# B&R Automation Studio project TD52 (part 19)

### mex.h
```c
/*
 * @(#)mex.h    generated by: makeheader 5.1.5  Tue May 24 21:10:37 2011
 *
 *		built from:	../../src/include/copyright.h
 *				../../src/include/pragma_interface.h
 *				mex_typedefs.h
 *				mexfunction.hpp
 *				fmexapi.cpp
 *				globals.cpp
 *				mexapi.cpp
 *				mexcbk.cpp
 *				mexdispatch.cpp
 *				mexintrf.cpp
 */

#if defined(_MSC_VER)
# pragma once
#endif
#if defined(__GNUC__) && (__GNUC__ > 3 || (__GNUC__ == 3 && __GNUC_MINOR__ > 3))
# pragma once
#endif

#ifndef mex_h
#define mex_h

/*
 * Copyright 1984-2003 The MathWorks, Inc.
 * All Rights Reserved.
 */

/* Copyright 2003-2006 The MathWorks, Inc. */

/* Only define EXTERN_C if it hasn't been defined already. This allows
 * individual modules to have more control over managing their exports.
 */
#ifndef EXTERN_C

#ifdef __cplusplus
  #define EXTERN_C extern "C"
#else
  #define EXTERN_C extern
#endif

#endif

/* Copyright 1999-2007 The MathWorks, Inc. */

/* $Revision: 1.7.4.4 $ */
#ifndef mex_typedefs_h
#define mex_typedefs_h

typedef struct impl_info_tag *MEX_impl_info;

#include "matrix.h"

#ifdef __cplusplus
extern "C"
{
#endif
typedef void (*mex_exit_fn)(void);
#ifdef __cplusplus
}
#endif

typedef struct mexGlobalTableEntry_Tag
{
    const char *name;             /* The name of the global */
    mxArray    **variable;        /* A pointer to the variable */
} mexGlobalTableEntry, *mexGlobalTable;

#ifdef _WIN32
#define cicompare(s1,s2) utStrcmpi((s1),(s2))
#else
#define cicompare(s1,s2) strcmp((s1),(s2))
#endif
#define cscompare(s1,s2) strcmp((s1),(s2))

typedef struct mexFunctionTableEntry_tag {
  const char *  name;
  mxFunctionPtr f;
  int           nargin;
  int           nargout;
  struct _mexLocalFunctionTable *local_function_table;
} mexFunctionTableEntry, *mexFunctionTable;

typedef struct _mexLocalFunctionTable {
  size_t           length;
  mexFunctionTable entries;
} _mexLocalFunctionTable, *mexLocalFunctionTable;

typedef struct {
  void (*initialize)(void);
  void (*terminate)(void);
} _mexInitTermTableEntry, *mexInitTermTableEntry;

#define MEX_INFORMATION_VERSION 1

typedef struct {
  int                   version;
  int                   file_function_table_length;
  mexFunctionTable      file_function_table;
  int                   global_variable_table_length;
  mexGlobalTable        global_variable_table;
  int                   npaths;
  const char **         paths;
  int                   init_term_table_length;
  mexInitTermTableEntry init_term_table;
} _mex_information, *mex_information;

typedef mex_information(*fn_mex_file)(void);

typedef void (*fn_clean_up_after_error)(void);
typedef const char *(*fn_simple_function_to_string)(mxFunctionPtr f);

typedef void (*fn_mex_enter_mex_library)(mex_information x);
typedef fn_mex_enter_mex_library fn_mex_exit_mex_library;

typedef mexLocalFunctionTable (*fn_mex_get_local_function_table)(void);
typedef mexLocalFunctionTable (*fn_mex_set_local_function_table)(mexLocalFunctionTable);

#endif

#ifdef DLL_EXPORT_SYM
# define MEXFUNCTION_LINKAGE EXTERN_C DLL_EXPORT_SYM
#else
# ifdef MW_NEEDS_VERSION_H
#  include "version.h"
#  define MEXFUNCTION_LINKAGE EXTERN_C DLL_EXPORT_SYM
# else
#  define MEXFUNCTION_LINKAGE EXTERN_C
# endif
#endif

MEXFUNCTION_LINKAGE
/*
 * mexFunction is the user-defined C routine that is called upon invocation
 * of a MEX-function.
 */
void mexFunction(
    int           nlhs,           /* number of expected outputs */
    mxArray       *plhs[],        /* array of pointers to output arguments */
    int           nrhs,           /* number of inputs */
    const mxArray *prhs[]         /* array of pointers to input arguments */
);

/*
 * This header file "mex.h" declares all the types, macros and
 * functions necessary to interface mex files with the current
 * version of MATLAB.  See the release notes for information on
 * supporting syntax from earlier versions.
 */
#include "matrix.h"

#include <stdio.h>

/*
 * Issue error message and return to MATLAB prompt
 */
EXTERN_C void mexErrMsgTxt(
    const char	*error_msg	/* string with error message */
    );

/*
 * Issue formatted error message with corresponding error identifier and return to MATLAB
 * prompt.
 */
EXTERN_C void mexErrMsgIdAndTxt(
    const char * identifier, /* string with error message identifier */
    const char * err_msg,    /* string with error message printf-style format */
    ...                      /* any additional arguments */
    );

/*
 * Invoke an unidentified warning. Such warnings can only be affected by the M-code
 * 'warning * all', since they have no specific identifier. See also mexWarnMsgIdAndTxt.
 */
EXTERN_C void mexWarnMsgTxt(
    const char	*warn_msg	/* string with warning message */
    );

/*
 * Invoke a warning with message identifier 'identifier' and message derived from 'fmt' and
 * subsequent arguments. The warning may either get printed as is (if it is set to 'on'), or
 * not actually get printed (if set to 'off'). See 'help warning' in MATLAB for more
 * details.
 */
EXTERN_C void mexWarnMsgIdAndTxt(
    const char * identifier,    /* string with warning message identifer */
    const char * warn_msg,	/* string with warning message printf-style format */
    ...                         /* any additional arguments */
    );

/*
 * mex equivalent to MATLAB's "disp" function
 */
EXTERN_C int mexPrintf(
    const char	*fmt,	/* printf style format */
    ...				/* any additional arguments */
    );

#define printf mexPrintf

/*
 * Remove all components of an array plus the array header itself
 * from MATLAB's memory allocation list.  The array will now
 * persist between calls to the mex function.  To destroy this
 * array, you will need to explicitly call mxDestroyArray().
 */
EXTERN_C void mexMakeArrayPersistent(
    mxArray *pa              /* pointer to array */
    );

/*
 * Remove memory previously allocated via mxCalloc from MATLAB's
 * memory allocation list.  To free this memory, you will need to
 * explicitly call mxFree().
 */
EXTERN_C void mexMakeMemoryPersistent(void *ptr);

/*
 * mex equivalent to MATLAB's "set" function
 */
EXTERN_C int mexSet(double handle, const char *property, mxArray *value);

/* API interface which mimics the "get" function */
EXTERN_C const mxArray *mexGet(double handle, const char *property);

/*
 * call MATLAB function
 */
EXTERN_C int mexCallMATLAB(
    int		nlhs,			/* number of expected outputs */
    mxArray	*plhs[],		/* pointer array to outputs */
    int		nrhs,			/* number of inputs */
    mxArray	*prhs[],		/* pointer array to inputs */
    const char	*fcn_name		/* name of function to execute */
    );

/*
 * call MATLAB function with Trap
 */
EXTERN_C mxArray	*mexCallMATLABWithTrap(
    int         nlhs,       /* number of expected outputs */
    mxArray     *plhs[],    /* pointer array to outputs */
    int         nrhs,       /* number of inputs */
    mxArray     *prhs[],    /* pointer array to inputs */
    const char  *fcn_name   /* name of function to execute */
    );

/*
 * set or clear mexCallMATLAB trap flag (if set then an error in
 * mexCallMATLAB is caught and mexCallMATLAB will return a status value,
 * if not set an error will cause control to revert to MATLAB)
 */
EXTERN_C void mexSetTrapFlag(int flag);

/*
 * Print an assertion-style error message and return control to the
 * MATLAB command line.
 */
EXTERN_C void mexPrintAssertion(
		const char *test,
		const char *fname,
		int linenum,
		const char *message);

/*
 * Tell whether or not a mxArray is in MATLAB's global workspace.
 */
EXTERN_C bool mexIsGlobal(const mxArray *pA);

/*
 * Place a copy of the array value into the specified workspace with the
 * specified name
 */
EXTERN_C int mexPutVariable(
    const char *workspace,
    const char *name,
    const mxArray *parray		/* matrix to copy */
    );

/*
 * return a pointer to the array value with the specified variable
 * name in the specified workspace
 */
EXTERN_C const mxArray *mexGetVariablePtr(
    const char *workspace,
    const char *name		/* name of symbol */
    );

/*
 * return a copy of the array value with the specified variable
 * name in the specified workspace
 */
EXTERN_C mxArray *mexGetVariable(
    const char	*workspace,
    const char  *name                /* name of variable in question */
    );

/*
 * Lock a MEX-function so that it cannot be cleared from memory.
 */
EXTERN_C void mexLock(void);

/*
 * Unlock a locked MEX-function so that it can be cleared from memory.
 */
EXTERN_C void mexUnlock(void);

/*
 * Return true if the MEX-function is currently locked, false otherwise.
 */
EXTERN_C bool mexIsLocked(void);

/*
 * Return the name of a the MEXfunction currently executing.
 */
EXTERN_C const char *mexFunctionName(void);

/*
 * Parse and execute MATLAB syntax in string.  Returns zero if successful,
 * and a non zero value if an error occurs.
 */
EXTERN_C int mexEvalString(
   const char *str	   /* matlab command string */
);

/*
 * Parse and execute MATLAB syntax in string.  Returns NULL if successful,
 * and an MException if an error occurs.
 */
EXTERN_C mxArray* mexEvalStringWithTrap(
   const char *str	   /* matlab command string */
);

/*
 * Register Mex-file's At-Exit function (accessed via MEX callback)
 */
EXTERN_C int mexAtExit(mex_exit_fn exit_fcn );

#endif /* mex_h */
```

### mwmathutil.h
```c
#if defined(_MSC_VER) || __GNUC__ > 3 || (__GNUC__ == 3 && __GNUC_MINOR__ > 3)
#pragma once
#endif

#ifndef mwmathutil_h
#define mwmathutil_h

/* Copyright 2003-2010 The MathWorks, Inc. */

/* Only define EXTERN_C if it hasn't been defined already. This allows
 * individual modules to have more control over managing their exports.
 */
#ifndef EXTERN_C

#ifdef __cplusplus
  #define EXTERN_C extern "C"
#else
  #define EXTERN_C extern
#endif

#endif

#include "tmwtypes.h"

/* abs(a) */
EXTERN_C double muDoubleScalarAbs(double a);

/* ceil(a) */
EXTERN_C double muDoubleScalarCeil(double a);

/* floor(a) */
EXTERN_C double muDoubleScalarFloor(double a);

/* round(a) */
EXTERN_C double muDoubleScalarRound(double a);

/* fix(a) */
EXTERN_C double muDoubleScalarFix(double xr);

/* acos(a) */
EXTERN_C double muDoubleScalarAcos(double a);

/* acosh(a) */
EXTERN_C double muDoubleScalarAcosh(double a);

/* asin(a) */
EXTERN_C double muDoubleScalarAsin(double a);

/* asinh(a) */
EXTERN_C double muDoubleScalarAsinh(double a);

/* atan(a) */
EXTERN_C double muDoubleScalarAtan(double a);

/* atanh(a) */
EXTERN_C double muDoubleScalarAtanh(double a);

/* cos(a) */
EXTERN_C double muDoubleScalarCos(double a);

/* cosh(a) */
EXTERN_C double muDoubleScalarCosh(double a);

/* exp(a) */
EXTERN_C double muDoubleScalarExp(double a);

/* log */
/*A warning 'Log of zero' should be issued by users for a = 0 */
EXTERN_C double muDoubleScalarLog(double a);

/* log10 */
/*A warning 'Log of zero' should be issued by users for a = 0 */
EXTERN_C double muDoubleScalarLog10(double a);

/* atan2(a,b) */
EXTERN_C double muDoubleScalarAtan2(double a, double b);

/* max(a,b) */
EXTERN_C double muDoubleScalarMax(double a, double b);

/* min(a,b) */
EXTERN_C double muDoubleScalarMin(double a, double b);

/* power(a,b) */
EXTERN_C double muDoubleScalarPower(double a, double b);

/* sin(a) */
EXTERN_C double muDoubleScalarSin(double a);

/* [s,c] = sincos(a) */
EXTERN_C void muDoubleScalarSinCos(double a, double* s, double* c);

/* sign(a) */
EXTERN_C double muDoubleScalarSign(double a);

/* sinh(a) */
EXTERN_C double muDoubleScalarSinh(double a);

/* sqrt(a) */
EXTERN_C double muDoubleScalarSqrt(double a);

/* tan(a) */
EXTERN_C double muDoubleScalarTan(double a);

/* tanh(a) */
EXTERN_C double muDoubleScalarTanh(double a);

/* mod(a,b) */
EXTERN_C double muDoubleScalarMod(double a, double b);

/* rem(a,b) */
EXTERN_C double muDoubleScalarRem(double a, double b);

/* hypot(a,b) */
EXTERN_C double muDoubleScalarHypot(double a,double b);

/* frexp(a,b) */
EXTERN_C double muDoubleScalarFrexp(double x, int *eptr);

/* abs(cmplx a) */
EXTERN_C double muDoubleComplexScalarAbs(double xr, double xi);

/* [br, bi] = exp(ar, ai) */
EXTERN_C void muDoubleComplexScalarExp(double *pyr, double *pyi, double xr, double xi);

/* hypot(ar, ai) */
EXTERN_C double muDoubleComplexScalarHypot(double ar, double ai, double br, double bi);

/* [br, bi] = log(ar, ai) */
EXTERN_C void muDoubleComplexScalarLog(double *pyr, double *pyi, double xr, double xi);

/* [cr, ci] = power(ar, ai, br, bi) */
EXTERN_C void muDoubleComplexScalarPower(double *cr, double *ci, double ar, double ai, double br, double bi);

/* [br, bi] = sqrt(ar, ai) */
EXTERN_C void muDoubleComplexScalarSqrt(double *br, double *bi, double ar, double ai);

/* [br, bi] = sign(ar, ai) */
EXTERN_C void muDoubleComplexScalarSign(double *br, double *bi, double ar, double ai);

/* [br, bi] = sin(ar, ai) */
EXTERN_C void muDoubleComplexScalarSin(double *br, double *bi, double ar, double ai);

/* [br, bi] = cos(ar, ai) */
EXTERN_C void muDoubleComplexScalarCos(double *br, double *bi, double ar, double ai);

/* [Sr, Si, Cr, Ci] = sincos(ar, ai) */
EXTERN_C void muDoubleComplexScalarSinCos(double *pySr, double *pySi, double *pyCr, double *pyCi,
                                          double xr, double xi);

/* [br, bi] = tan(ar, ai) */
EXTERN_C void muDoubleComplexScalarTan(double *br, double *bi, double ar, double ai);

/* [br, bi] = atan(ar, ai) */
EXTERN_C void muDoubleComplexScalarAtan(double *br, double *bi, double ar, double ai);

/* [br, bi] = asin(ar, ai) */
EXTERN_C void muDoubleComplexScalarAsin(double *br, double *bi, double ar, double ai);

/* [br, bi] = acos(ar, ai) */
EXTERN_C void muDoubleComplexScalarAcos(double *br, double *bi, double ar, double ai);

/* [br, bi] = sinh(ar, ai) */
EXTERN_C void muDoubleComplexScalarSinh(double *br, double *bi, double ar, double ai);

/* [br, bi] = cosh(ar, ai) */
EXTERN_C void muDoubleComplexScalarCosh(double *br, double *bi, double ar, double ai);

/* [br, bi] = tanh(ar, ai) */
EXTERN_C void muDoubleComplexScalarTanh(double *br, double *bi, double ar, double ai);

/* [br, bi] = asinh(ar, ai) */
EXTERN_C void muDoubleComplexScalarAsinh(double *br, double *bi, double ar, double ai);

/* [br, bi] = acosh(ar, ai) */
EXTERN_C void muDoubleComplexScalarAcosh(double *br, double *bi, double ar, double ai);

/* Single-precision functions */

/* abs(a) */
EXTERN_C float muSingleScalarAbs(float a);

/* ceil(a) */
EXTERN_C float muSingleScalarCeil(float a);

/* floor(a) */
EXTERN_C float muSingleScalarFloor(float a);

/* round(a) */
EXTERN_C float muSingleScalarRound(float a);

/* fix(a) */
EXTERN_C float muSingleScalarFix(float xr);

/* acos(a) */
EXTERN_C float muSingleScalarAcos(float a);

/* acosh(a) */
EXTERN_C float muSingleScalarAcosh(float a);

/* asin(a) */
EXTERN_C float muSingleScalarAsin(float a);

/* asinh(a) */
EXTERN_C float muSingleScalarAsinh(float a);

/* atan(a) */
EXTERN_C float muSingleScalarAtan(float a);

/* atanh(a) */
EXTERN_C float muSingleScalarAtanh(float a);

/* cos(a) */
EXTERN_C float muSingleScalarCos(float a);

/* cosh(a) */
EXTERN_C float muSingleScalarCosh(float a);

/* exp(a) */
EXTERN_C float muSingleScalarExp(float a);

/* log */
/*A warning 'Log of zero' should be issued by users for a = 0 */
EXTERN_C float muSingleScalarLog(float a);

/* log10 */
/*A warning 'Log of zero' should be issued by users for a = 0 */
EXTERN_C float muSingleScalarLog10(float a);

/* atan2(a,b) */
EXTERN_C float muSingleScalarAtan2(float a, float b);

/* max(a,b) */
EXTERN_C float muSingleScalarMax(float a, float b);

/* min(a,b) */
EXTERN_C float muSingleScalarMin(float a, float b);

/* power(a,b) */
EXTERN_C float muSingleScalarPower(float a, float b);

/* sin(a) */
EXTERN_C float muSingleScalarSin(float a);

/* [s,c] = sincos(a) */
EXTERN_C void muSingleScalarSinCos(float a, float* s, float* c);

/* sign(a) */
EXTERN_C float muSingleScalarSign(float a);

/* sinh(a) */
EXTERN_C float muSingleScalarSinh(float a);

/* sqrt(a) */
EXTERN_C float muSingleScalarSqrt(float a);

/* tan(a) */
EXTERN_C float muSingleScalarTan(float a);

/* tanh(a) */
EXTERN_C float muSingleScalarTanh(float a);

/* mod(a,b) */
EXTERN_C float muSingleScalarMod(float a, float b);

/* rem(a,b) */
EXTERN_C float muSingleScalarRem(float a, float b);

/* hypot(a,b) */
EXTERN_C float muSingleScalarHypot(float a,float b);

/* frexp(a,b) */
EXTERN_C float muSingleScalarFrexp(float x, int *eptr);

/* abs(cmplx a) */
EXTERN_C float muSingleComplexScalarAbs(float xr, float xi);

/* [br, bi] = exp(ar, ai) */
EXTERN_C void muSingleComplexScalarExp(float *pyr, float *pyi, float xr, float xi);

/* hypot(ar, ai) */
EXTERN_C float muSingleComplexScalarHypot(float ar, float ai, float br, float bi);

/* [br, bi] = log(ar, ai) */
EXTERN_C void muSingleComplexScalarLog(float *pyr, float *pyi, float xr, float xi);

/* [cr, ci] = power(ar, ai, br, bi) */
EXTERN_C void muSingleComplexScalarPower(float *cr, float *ci, float ar, float ai, float br, float bi);

/* [br, bi] = sqrt(ar, ai) */
EXTERN_C void muSingleComplexScalarSqrt(float *br, float *bi, float ar, float ai);

/* [br, bi] = sign(ar, ai) */
EXTERN_C void muSingleComplexScalarSign(float *br, float *bi, float ar, float ai);

/* [br, bi] = sin(ar, ai) */
EXTERN_C void muSingleComplexScalarSin(float *br, float *bi, float ar, float ai);

/* [br, bi] = cos(ar, ai) */
EXTERN_C void muSingleComplexScalarCos(float *br, float *bi, float ar, float ai);

/* [Sr, Si, Cr, Ci] = sincos(ar, ai) */
EXTERN_C void muSingleComplexScalarSinCos(float *pySr, float *pySi, float *pyCr, float *pyCi,
                                          float xr, float xi);

/* [br, bi] = tan(ar, ai) */
EXTERN_C void muSingleComplexScalarTan(float *br, float *bi, float ar, float ai);

/* [br, bi] = atan(ar, ai) */
EXTERN_C void muSingleComplexScalarAtan(float *br, float *bi, float ar, float ai);

/* [br, bi] = asin(ar, ai) */
EXTERN_C void muSingleComplexScalarAsin(float *br, float *bi, float ar, float ai);

/* [br, bi] = acos(ar, ai) */
EXTERN_C void muSingleComplexScalarAcos(float *br, float *bi, float ar, float ai);

/* [br, bi] = sinh(ar, ai) */
EXTERN_C void muSingleComplexScalarSinh(float *br, float *bi, float ar, float ai);

/* [br, bi] = cosh(ar, ai) */
EXTERN_C void muSingleComplexScalarCosh(float *br, float *bi, float ar, float ai);

/* [br, bi] = tanh(ar, ai) */
EXTERN_C void muSingleComplexScalarTanh(float *br, float *bi, float ar, float ai);

/* [br, bi] = asinh(ar, ai) */
EXTERN_C void muSingleComplexScalarAsinh(float *br, float *bi, float ar, float ai);

/* [br, bi] = acosh(ar, ai) */
EXTERN_C void muSingleComplexScalarAcosh(float *br, float *bi, float ar, float ai);

#ifdef __WATCOMC__
#pragma aux muDoubleScalarAbs value [8087];
#pragma aux muDoubleScalarCeil value [8087];
#pragma aux muDoubleScalarFloor value [8087];
#pragma aux muDoubleScalarRound value [8087];
#pragma aux muDoubleScalarAcos value [8087];
#pragma aux muDoubleScalarAcosh value [8087];
#pragma aux muDoubleScalarAsin value [8087];
#pragma aux muDoubleScalarAsinh value [8087];
#pragma aux muDoubleScalarAtan value [8087];
#pragma aux muDoubleScalarAtanh value [8087];
#pragma aux muDoubleScalarCos value [8087];
#pragma aux muDoubleScalarCosh value [8087];
#pragma aux muDoubleScalarExp value [8087];
#pragma aux muDoubleScalarLog value [8087];
#pragma aux muDoubleScalarLog10 value [8087];
#pragma aux muDoubleScalarAtan2 value [8087]
#pragma aux muDoubleScalarMax value [8087]
#pragma aux muDoubleScalarMin value [8087]
#pragma aux muDoubleScalarPower value [8087]
#pragma aux muDoubleScalarSin value [8087];
#pragma aux muDoubleScalarSinCos value [8087];
#pragma aux muDoubleScalarSign value [8087];
#pragma aux muDoubleScalarSinh value [8087];
#pragma aux muDoubleScalarSqrt value [8087];
#pragma aux muDoubleScalarTan value [8087];
#pragma aux muDoubleScalarTanh value [8087];
#pragma aux muDoubleScalarMod value [8087]
#pragma aux muDoubleScalarRem value [8087]
#pragma aux muDoubleScalarHypot value [8087];
#pragma aux muDoubleScalarFix value [8087];
#pragma aux muDoubleScalarFrexp value [8087];
#pragma aux muDoubleComplexScalarAbs value [8087];
#pragma aux muDoubleComplexScalarExp value [8087];
#pragma aux muDoubleComplexScalarHypot value [8087];
#pragma aux muDoubleComplexScalarLog value [8087];
#pragma aux muDoubleComplexScalarPower value [8087];
#pragma aux muDoubleComplexScalarSqrt value [8087];
#pragma aux muDoubleComplexScalarSign value [8087];
#pragma aux muDoubleComplexScalarSin value [8087];
#pragma aux muDoubleComplexScalarCos value [8087];
#pragma aux muDoubleComplexScalarSinCos value [8087];
#pragma aux muDoubleComplexScalarTan value [8087];
#pragma aux muDoubleComplexScalarAtan value [8087];
#pragma aux muDoubleComplexScalarAsin value [8087];
#pragma aux muDoubleComplexScalarAcos value [8087];
#pragma aux muDoubleComplexScalarSinh value [8087];
#pragma aux muDoubleComplexScalarCosh value [8087];
#pragma aux muDoubleComplexScalarTanh value [8087];
#pragma aux muDoubleComplexScalarAsinh value [8087];
#pragma aux muDoubleComplexScalarAcosh value [8087];
#pragma aux muSingleScalarAbs value [8087];
#pragma aux muSingleScalarCeil value [8087];
#pragma aux muSingleScalarFloor value [8087];
#pragma aux muSingleScalarRound value [8087];
#pragma aux muSingleScalarAcos value [8087];
#pragma aux muSingleScalarAcosh value [8087];
#pragma aux muSingleScalarAsin value [8087];
#pragma aux muSingleScalarAsinh value [8087];
#pragma aux muSingleScalarAtan value [8087];
#pragma aux muSingleScalarAtanh value [8087];
#pragma aux muSingleScalarCos value [8087];
#pragma aux muSingleScalarCosh value [8087];
#pragma aux muSingleScalarExp value [8087];
#pragma aux muSingleScalarLog value [8087];
#pragma aux muSingleScalarLog10 value [8087];
#pragma aux muSingleScalarAtan2 value [8087]
#pragma aux muSingleScalarMax value [8087]
#pragma aux muSingleScalarMin value [8087]
#pragma aux muSingleScalarPower value [8087]
#pragma aux muSingleScalarSin value [8087];
#pragma aux muSingleScalarSinCos value [8087];
#pragma aux muSingleScalarSign value [8087];
#pragma aux muSingleScalarSinh value [8087];
#pragma aux muSingleScalarSqrt value [8087];
#pragma aux muSingleScalarTan value [8087];
#pragma aux muSingleScalarTanh value [8087];
#pragma aux muSingleScalarMod value [8087]
#pragma aux muSingleScalarRem value [8087]
#pragma aux muSingleScalarHypot value [8087];
#pragma aux muSingleScalarFix value [8087];
#pragma aux muSingleScalarFrexp value [8087];
#pragma aux muSingleComplexScalarAbs value [8087];
#pragma aux muSingleComplexScalarExp value [8087];
#pragma aux muSingleComplexScalarHypot value [8087];
#pragma aux muSingleComplexScalarLog value [8087];
#pragma aux muSingleComplexScalarPower value [8087];
#pragma aux muSingleComplexScalarSqrt value [8087];
#pragma aux muSingleComplexScalarSign value [8087];
#pragma aux muSingleComplexScalarSin value [8087];
#pragma aux muSingleComplexScalarCos value [8087];
#pragma aux muSingleComplexScalarSinCos value [8087];
#pragma aux muSingleComplexScalarTan value [8087];
#pragma aux muSingleComplexScalarAtan value [8087];
#pragma aux muSingleComplexScalarAsin value [8087];
#pragma aux muSingleComplexScalarAcos value [8087];
#pragma aux muSingleComplexScalarSinh value [8087];
#pragma aux muSingleComplexScalarCosh value [8087];
#pragma aux muSingleComplexScalarTanh value [8087];
#pragma aux muSingleComplexScalarAsinh value [8087];
#pragma aux muSingleComplexScalarAcosh value [8087];
#endif

/* Integer Scalar functions. */
/* Integer Abs Family. */
EXTERN_C uint8_T muIntScalarAbs_uint8(uint8_T a);

EXTERN_C int8_T muIntScalarAbs_sint8(int8_T a);

EXTERN_C uint16_T muIntScalarAbs_uint16(uint16_T a);

EXTERN_C int16_T muIntScalarAbs_sint16(int16_T a);

EXTERN_C uint32_T muIntScalarAbs_uint32(uint32_T a);

EXTERN_C int32_T muIntScalarAbs_sint32(int32_T a);

/* Integer Max Family. */
EXTERN_C uint8_T muIntScalarMax_uint8(uint8_T a, uint8_T b);

EXTERN_C int8_T muIntScalarMax_sint8(int8_T a, int8_T b);

EXTERN_C uint16_T muIntScalarMax_uint16(uint16_T a, uint16_T b);

EXTERN_C int16_T muIntScalarMax_sint16(int16_T a, int16_T b);

EXTERN_C uint32_T muIntScalarMax_uint32(uint32_T a, uint32_T b);

EXTERN_C int32_T muIntScalarMax_sint32(int32_T a, int32_T b);

/* Integer Min Family. */
EXTERN_C uint8_T muIntScalarMin_uint8(uint8_T a, uint8_T b);

EXTERN_C int8_T muIntScalarMin_sint8(int8_T a, int8_T b);

EXTERN_C uint16_T muIntScalarMin_uint16(uint16_T a, uint16_T b);

EXTERN_C int16_T muIntScalarMin_sint16(int16_T a, int16_T b);

EXTERN_C uint32_T muIntScalarMin_uint32(uint32_T a, uint32_T b);

EXTERN_C int32_T muIntScalarMin_sint32(int32_T a, int32_T b);

/* Integer Mod Family. */
EXTERN_C uint8_T muIntScalarMod_uint8(uint8_T a, uint8_T b);

EXTERN_C int8_T muIntScalarMod_sint8(int8_T a, int8_T b);

EXTERN_C uint16_T muIntScalarMod_uint16(uint16_T a, uint16_T b);

EXTERN_C int16_T muIntScalarMod_sint16(int16_T a, int16_T b);

EXTERN_C uint32_T muIntScalarMod_uint32(uint32_T a, uint32_T b);

EXTERN_C int32_T muIntScalarMod_sint32(int32_T a, int32_T b);

/* Integer Rem Family. */
EXTERN_C uint8_T muIntScalarRem_uint8(uint8_T a, uint8_T b);

EXTERN_C int8_T muIntScalarRem_sint8(int8_T a, int8_T b);

EXTERN_C uint16_T muIntScalarRem_uint16(uint16_T a, uint16_T b);

EXTERN_C int16_T muIntScalarRem_sint16(int16_T a, int16_T b);

EXTERN_C uint32_T muIntScalarRem_uint32(uint32_T a, uint32_T b);

EXTERN_C int32_T muIntScalarRem_sint32(int32_T a, int32_T b);

/* Integer Sign Family. */
EXTERN_C uint8_T muIntScalarSign_uint8(uint8_T a);

EXTERN_C int8_T muIntScalarSign_sint8(int8_T a);

EXTERN_C uint16_T muIntScalarSign_uint16(uint16_T a);

EXTERN_C int16_T muIntScalarSign_sint16(int16_T a);

EXTERN_C uint32_T muIntScalarSign_uint32(uint32_T a);

EXTERN_C int32_T muIntScalarSign_sint32(int32_T a);

/* isFinite(a) */
EXTERN_C boolean_T muDoubleScalarIsFinite(double a);

/* isNaN(a) */
EXTERN_C boolean_T muDoubleScalarIsNaN(double a);

/* isInf(a) */
EXTERN_C boolean_T muDoubleScalarIsInf(double a);

/* isFinite(ar, ai) */
EXTERN_C boolean_T muDoubleComplexScalarIsFinite(double ar, double ai);

/* isNaN(a) */
EXTERN_C boolean_T muDoubleComplexScalarIsNaN(double ar, double ai);

/* isInf(ar, ai) */
EXTERN_C boolean_T muDoubleComplexScalarIsInf(double ar, double ai);

/* Single-precision functions */

/* isFinite(a) */
EXTERN_C boolean_T muSingleScalarIsFinite(float a);

/* isNaN(a) */
EXTERN_C boolean_T muSingleScalarIsNaN(float a);

/* isInf(a) */
EXTERN_C boolean_T muSingleScalarIsInf(float a);

/* isFinite(ar, ai) */
EXTERN_C boolean_T muSingleComplexScalarIsFinite(float ar, float ai);

/* isNaN(a) */
EXTERN_C boolean_T muSingleComplexScalarIsNaN(float ar, float ai);

/* isInf(ar, ai) */
EXTERN_C boolean_T muSingleComplexScalarIsInf(float ar, float ai);

#endif /* mwmathutil_h */
```

### mwutil.h
```c
/*
 * @(#)mwutil.h    generated by: makeheader 5.1.5  Tue May 24 21:07:18 2011
 *
 *		built from:	../../src/include/copyright.h
 *				../../src/include/pragma_interface.h
 *				cputime.cpp
 *				cycles.cpp
 *				dconvert.cpp
 *				demangle.cpp
 *				dynload.cpp
 *				emptystr.cpp
 *				enum_str.cpp
 *				expmatch.cpp
 *				f2cstr.cpp
 *				fgets.cpp
 *				filelink.cpp
 *				format.cpp
 *				fp_conv.cpp
 *				fpu.cpp
 *				getcwd.cpp
 *				hash.cpp
 *				incrfcn.cpp
 *				int_conv.cpp
 *				logfile.cpp
 *				lower.cpp
 *				multibyte.cpp
 *				mwclasses.cpp
 *				perfcount.cpp
 *				printf.cpp
 *				purifytools.cpp
 *				set.cpp
 *				special_nans.cpp
 *				stacktrc.cpp
 *				strcat.cpp
 *				strcmp.cpp
 *				strcmpi.cpp
 *				strcpy.cpp
 *				strdup.cpp
 *				strlen.cpp
 *				strrep.cpp
 *				strrstr.cpp
 *				strtok.cpp
 *				sysinfo.cpp
 *				timeinfo.cpp
 *				tmpnam.cpp
 *				tolower.cpp
 *				upper.cpp
 *				utStreamUtilities.cpp
 *				ut_alloca.cpp
 *				utassert.cpp
 *				utcrc.cpp
 *				utsignal.cpp
 *				wallclok.cpp
 *				array/array.cpp
 *				basic/basic_contexts.cpp
 *				checksum/md5checksum.cpp
 *				coll/functional.cpp
 *				coll/hash_map.cpp
 *				coll/hashrank.cpp
 *				cpputils/attacher.cpp
 *				cpputils/chunkedptr.cpp
 *				cpputils/countlist.cpp
 *				cpputils/safepointer.cpp
 *				cpputils/stat_ref_ok.cpp
 *				cpputils/stl_allocator.cpp
 *				dsbuffer/dsbuffer.cpp
 *				dtoa/dtoa.cpp
 *				dtoa/fpc.cpp
 *				dtoa/g_fmt.cpp
 *				err/error_context.cpp
 *				except/cmnHooks.cpp
 *				except/cmnSystemCalls.cpp
 *				except/errInternalException.cpp
 *				except/errSystemError.cpp
 *				except/errThrowable.cpp
 *				except/errUserException.cpp
 *				except/exceptCleanup.cpp
 *				except/exceptTypedefs.cpp
 *				except/instCpuCounter.cpp
 *				except/instInstrument.cpp
 *				except/instStopwatch.cpp
 *				except/logBasicSystemHandler.cpp
 *				except/logDataOutput.cpp
 *				except/logDebugOutputHandler.cpp
 *				except/logExternalizable.cpp
 *				except/logFilter.cpp
 *				except/logFormattable.cpp
 *				except/logFormatter.cpp
 *				except/logHandler.cpp
 *				except/logLevel.cpp
 *				except/logLogger.cpp
 *				except/logObjectOutput.cpp
 *				except/logObjectOutputStream.cpp
 *				except/logOutputStreamHandler.cpp
 *				except/logStreamHandler.cpp
 *				except/logTerminalHandler.cpp
 *				except/logXmlFormatter.cpp
 *				except/msgMsgCodeException.cpp
 *				except/msgMsgFormat.cpp
 *				except/usrReport.cpp
 *				except/usrRunning.cpp
 *				except/usrStartup.cpp
 *				except/usrStrategy.cpp
 *				ghash/ghash.cpp
 *				gtable/gtable.cpp
 *				hashtool/hashtool.cpp
 *				icuext/uchar.cpp
 *				icuext/uconv.cpp
 *				icuext/uctype.cpp
 *				icuext/uerror.cpp
 *				icuext/uhash.cpp
 *				icuext/umisc.cpp
 *				icuext/urecognize.cpp
 *				icuext/uspecial.cpp
 *				icuext/ustdio.cpp
 *				icuext/ustring.cpp
 *				icuext/utf.cpp
 *				icuext/utf8str.cpp
 *				ihash/ihash.cpp
 *				interval/fsi.cpp
 *				lcctype/utctype.cpp
 *				linebuf/linebuf.cpp
 *				mem/memory_context.cpp
 *				memmgr/memalloc.cpp
 *				msg/message_context.cpp
 *				nh/namehash.cpp
 *				nh/symtab.cpp
 *				profile/profile.cpp
 *				regexp/re_api.cpp
 *				regexp/re_builder.cpp
 *				regexp/re_collection.cpp
 *				regexp/re_context.cpp
 *				regexp/re_evaluator.cpp
 *				regexp/re_flags.cpp
 *				regexp/re_memory.cpp
 *				regexp/re_node_factory.cpp
 *				regexp/re_parser.cpp
 *				regexp/re_parser_context.cpp
 *				regexp/re_private_nodes.cpp
 *				regexp/re_protected_nodes.cpp
 *				regexp/re_replace.cpp
 *				regexp/re_replace_nodes.cpp
 *				regexp/re_replace_parser.cpp
 *				regexp/re_replaceable.cpp
 *				regexp/re_results.cpp
 *				regexp/re_search_info.cpp
 *				regexp/re_token_info.cpp
 *				regexp/re_translate.cpp
 *				regexp/re_tree.cpp
 *				regexp/re_tree_parser.cpp
 *				regexp/re_util.cpp
 *				sort/qsort.cpp
 *				strbuf/string_buffer.cpp
 *				threads/atomic.cpp
 *				threads/mwatomic.cpp
 *				threads/mwbarrier.cpp
 *				threads/mwconcurrent.cpp
 *				threads/mwcondition.cpp
 *				threads/mwcountedbody.cpp
 *				threads/mwcountedpointer.cpp
 *				threads/mwevent.cpp
 *				threads/mwmonitor.cpp
 *				threads/mwmutex_lwm.cpp
 *				threads/mwmutexlock.cpp
 *				threads/mwobjmgr.cpp
 *				threads/mwpointer.cpp
 *				threads/mwrcrsvmtx.cpp
 *				threads/mwsemaphore.cpp
 *				threads/mwsingleton.cpp
 *				threads/mwthdspc.cpp
 *				threads/mwthread.cpp
 *				threads/mwthreadid.cpp
 *				threads/mwtimeunit.cpp
 *				threads/ut_thread.cpp
 *				tse/tse.cpp
 *				warn/warning_context.cpp
 *				warn/warnmgr.cpp
 */

#if defined(_MSC_VER)
# pragma once
#endif
#if defined(__GNUC__) && (__GNUC__ > 3 || (__GNUC__ == 3 && __GNUC_MINOR__ > 3))
# pragma once
#endif

#ifndef mwutil_h
#define mwutil_h

/*
 * Copyright 1984-2003 The MathWorks, Inc.
 * All Rights Reserved.
 */

/* Copyright 2003-2006 The MathWorks, Inc. */

/* Only define EXTERN_C if it hasn't been defined already. This allows
 * individual modules to have more control over managing their exports.
 */
#ifndef EXTERN_C

#ifdef __cplusplus
  #define EXTERN_C extern "C"
#else
  #define EXTERN_C extern
#endif

#endif

/*
 * load library into memory
 */
EXTERN_C void *utLoadLibrary(
    const char	*fullname,	/* _full_ library path name */
    int		*errorStatus	/* return variable for error code */
    );

/*
 * Check whether shared library is loaded without loading it
 * Takes basename. Returns true if the library is loaded
 */
EXTERN_C bool utIsLibraryLoaded(const char *name);

/*
 * Return handle for already loaded library
 */
EXTERN_C void *utLoadModule(const char *basename);

/*
 * lookup symbol in a loaded library
 */
EXTERN_C void *utFindSymbolInLibrary(
    void        *handle,	/* handle returned by utLoadLibrary */
    const char  *symbol         /* symbol name to look up */
    );

/*
 * unload a previously loaded library
 */
EXTERN_C int utUnloadLibrary(
    void        *handle		/* handle returned by utLoadLibrary */
    );

/*
 * Retrieve last error in dynamic loader utility routines
 */
EXTERN_C const char *utLastLibraryError(void);

/*
 * Predicate to determine whether a double is an int.
 * -0 is not considered an int, because converting it back
 * does not yield the same double.
 */
EXTERN_C bool utDblIsInt(double x);

/*
 * Use unique NaNs as flags for special values
 * These values should never be generated by Matlab as valid NaNs.
 *
 * The low-order word is all zeros.
 */

#define UT_SPECIAL_NAN 0x7ff5c5c0

#define UT_NAN_NEVER_TOUCHED (UT_SPECIAL_NAN + 0x1)
#define UT_NAN_FORLOOP_EMPTY (UT_SPECIAL_NAN + 0x2)

#define UT_SET_NAN_VALUE(lval, jqnan) ut_SET_BOTH(lval, jqnan, 0)

/*
 * since the x86 fpu can change the leading mastissa bit on QNaNs, we check for
 * equality with and without the bit set.
 */
#define UT_QNAN_BITMASK 0x00080000
#define UT_IS_NAN_VALUE(val, jqnan)                                                                     \
    (*(((int*)&(val))+(CPU_NUM_FORMAT==FIEEE_BE)) == 0x0 &&                                             \
     (*(((int*)&(val))+(CPU_NUM_FORMAT==FIEEE_LE))|UT_QNAN_BITMASK) == ((jqnan)|UT_QNAN_BITMASK))

# define utAssert(test)             ((void)0)
# define utAssertStr(test, message) ((void)0)
# define utAssertAlways(message)    ((void)0)

#endif /* mwutil_h */
```

### odesup.h
```c
/*
 * Copyright 1994-2008 The MathWorks, Inc.
 *
 * File: odesup.h     $Revision: 1.3.4.3 $
 *
 * Abstract:
 *
 */

#ifndef __ODE_SUP__
#define __ODE_SUP__

#include <math.h>
#include <stddef.h> /* needed for NULL */

#include "tmwtypes.h"

#ifdef RT_MALLOC
# include <stdlib.h>
#endif

#ifdef USE_RTMODEL
# include "simstruc_types.h"
#else
# include "simstruc.h"
#endif

#ifndef RT_MALLOC
# ifndef NCSTATES
#  error "must define NCSTATES"
# endif
#endif

extern const char *RT_MEMORY_ALLOCATION_ERROR;

#ifdef RT_MALLOC
# define DERIVATIVES(si) rtmiDerivatives(*rtsiGetModelMethodsPtr(si))
# define PROJECTION(si)  rtmiProjection(*rtsiGetModelMethodsPtr(si))
# define OUTPUTS(si,tid) rtmiOutputs(*rtsiGetModelMethodsPtr(si),tid)
#else
# define DERIVATIVES(si) MdlDerivatives()
# define OUTPUTS(si,tid) MdlOutputs(tid)
# define PROJECTION(si)  MdlProjection()
  extern void MdlDerivatives(void);
  extern void MdlOutputs(int_T tid);
  extern void MdlProjection(void);
#endif

#ifndef USE_RTMODEL

void rt_ODECreateIntegrationData(RTWSolverInfo *si);
void rt_ODEDestroyIntegrationData(RTWSolverInfo *si);
void rt_ODEUpdateContinuousStates(RTWSolverInfo *si);

void rt_ODECacheDataIntoSolverInfo(SimStruct *S)
{
    RTWSolverInfo *si = ssGetRTWSolverInfo(S);

    if (si != NULL) {
        rtsiSetSolverStopTime(si, ssGetSolverStopTime(S));
        rtsiSetSolverName(si, ssGetSolverName(S));
        rtsiSetSolverData(si, ssGetSolverData(S));
    }
}

void rt_ODERetrieveDataFromSolverInfo(SimStruct *S)
{
    RTWSolverInfo *si = ssGetRTWSolverInfo(S);

    if (si != NULL) {
        ssSetSolverStopTime(S, rtsiGetSolverStopTime(si));
        ssSetSolverData(S, rtsiGetSolverData(si));
        ssSetSolverName(S, rtsiGetSolverName(si));
    }
}

const char_T *rt_ODECreateSolverInfo(SimStruct *S)
{
    const char_T          *errStatus = NULL;
    RTWSolverInfo         *si        = NULL;
    RTWRTModelMethodsInfo *mmi       = NULL;

#ifndef RT_MALLOC
    static RTWSolverInfo _si;
    static RTWRTModelMethodsInfo _mdlMths;

    si  = &_si;
    mmi = &_mdlMths;
#else
    si = (RTWSolverInfo *)malloc(sizeof(RTWSolverInfo));
    if (si == NULL) {
        errStatus = RT_MEMORY_ALLOCATION_ERROR;
        ssSetErrorStatus(S, RT_MEMORY_ALLOCATION_ERROR);
        goto EXIT_POINT;
    }

    mmi = (RTWRTModelMethodsInfo *)malloc(sizeof(RTWRTModelMethodsInfo));
    if (mmi == NULL) {
        errStatus = RT_MEMORY_ALLOCATION_ERROR;
        ssSetErrorStatus(S, RT_MEMORY_ALLOCATION_ERROR);
        goto EXIT_POINT;
    }
#endif

    rtsiSetModelMethodsPtr(si, mmi);
    rtsiSetRTModelPtr(si, (void *)S);
    rtmiSetRTModelPtr(*mmi, (void *)S);

    ssSetRTWSolverInfo(S, si);

    /*
     * The fields below need to be copied over at setup
     * and copied back into the SimStruct at the end
     */
    rt_ODECacheDataIntoSolverInfo(S);

    /*
     * The fields below only need to be setup. They are
     * pointer fields and updating them will automatically
     * update the owner SimStruct
     */

    /* Copy over a pointer to StepSize */
    rtsiSetStepSizePtr(si, &ssGetStepSize(S));

    /* Copy over a pointer to SimTimeStep */
    rtsiSetSimTimeStepPtr(si, &ssGetSimTimeStep(S));

    /* Copy over a pointer to the time pointer */
    rtsiSetTPtr(si, &ssGetTPtr(S));

    /* Copy over a pointer to the location of the derivs */
    rtsiSetdXPtr(si, &ssGetdX(S));

    /* Copy over a pointer to the location of the cont states */
    rtsiSetContStatesPtr(si, &ssGetContStates(S));

    /* Copy over a pointer to the location of the number of cont states */
    rtsiSetNumContStatesPtr(si, &ssGetNumContStates(S));

    /* Copy over a pointer to the location of the error status */
    rtsiSetErrorStatusPtr(si, &ssGetErrorStatus(S));

    /* Copy over the order of extrapolation method */
    rtsiSetSolverExtrapolationOrder(si, ssGetSolverExtrapolationOrder(S));

    /* Copy over the number of Newton iterations */
    rtsiSetSolverNumberNewtonIterations(si, ssGetSolverNumberNewtonIterations(S));

#ifdef RT_MALLOC
  EXIT_POINT:
#endif
    return(errStatus);
}

void rt_CreateIntegrationData(SimStruct *S)
{
    if (rt_ODECreateSolverInfo(S) != NULL) {
        return;
    }

    rt_ODECreateIntegrationData(ssGetRTWSolverInfo(S));

    rt_ODERetrieveDataFromSolverInfo(S);
}

#ifdef RT_MALLOC
void rt_DestroyIntegrationData(SimStruct *S)
{
    RTWSolverInfo *si = NULL;

    rt_ODECacheDataIntoSolverInfo(S);

    si = ssGetRTWSolverInfo(S);

    if (si != NULL) {
        rt_ODEDestroyIntegrationData(si);
        free(rtsiGetModelMethodsPtr(si));
        free(si);
        ssSetRTWSolverInfo(S, NULL);
    }
}
#endif

void rt_UpdateContinuousStates(SimStruct *S)
{
    rt_ODECacheDataIntoSolverInfo(S);
    rt_ODEUpdateContinuousStates(ssGetRTWSolverInfo(S));
    rt_ODERetrieveDataFromSolverInfo(S);
}

#endif
#endif /* __ODE_SUP__ */
```

### pt_info.h
```c
/*
 * Copyright 1994-2002 The MathWorks, Inc.
 *
 * File: pt_info.h     $Revision: 1.13 $
 *
 * Abstract:
 *   Parameter tuning information.  For details about these structures
 *   see MATLAB/rtw/c/src/pt_readme.txt.
 */

#ifndef __PT_INFO__
#define __PT_INFO__

#include <tmwtypes.h>

typedef enum {
    rt_SCALAR,
    rt_VECTOR,
    rt_MATRIX_ROW_MAJOR,
    rt_MATRIX_COL_MAJOR,
    rt_MATRIX_COL_MAJOR_ND
} ParamClass;

typedef enum {
    rt_SL_PARAM,
    rt_SF_PARAM,
    rt_SHARED_PARAM
} ParamSource;

typedef struct ParameterTuning_tag {
    ParamClass  paramClass;   /* Class of parameter               */
    int_T       nRows;        /* Number of rows                   */
    int_T       nCols;        /* Number of columns                */
    int_T       nDims;        /* Number of dimensions             */
    int_T       dimsOffset;   /* Offset into dimensions vector    */
    ParamSource source;       /* Source of parameter              */
    uint_T      dataType;     /* data type enumeration            */
    uint_T      numInstances; /* Number of parameter instances    */
    int_T       mapOffset;    /* Offset into map vector           */
} ParameterTuning;

typedef struct BlockTuning_tag {
    const char_T      *blockName;   /* Block name                       */
    const char_T      *paramName;   /* Parameter name                   */
    ParameterTuning    ptRec;       /* Parameter tuning record          */
} BlockTuning;

typedef struct VariableTuning_tag {
    const char_T *varName;    /* Variable name                    */
    ParameterTuning ptRec;    /* Parameter tuning record          */
} VariableTuning;

#define ptinfoGetClass(pt)            (pt)->paramClass
#define ptinfoGetNumRows(pt)          (pt)->nRows
#define ptinfoGetNumCols(pt)          (pt)->nCols
#define ptinfoGetNumDimensions(pt)    (pt)->nDims
#define ptinfoGetSource(pt)           (pt)->source
#define ptinfoGetDataTypeEnum(pt)     (pt)->dataType
#define ptinfoGetNumInstances(pt)     (pt)->numInstances
#define ptinfoGetParametersOffset(pt) (pt)->mapOffset
#define ptinfoGetDimensionsOffset(pt) (pt)->dimsOffset

#endif  /* __PT_INFO__ */
```

### rt_logging.h
```c
/*
 * @(#)rt_logging.h    generated by: makeheader 5.1.5  Tue May 24 21:25:56 2011
 *
 *		built from:	rt_logging.c
 */

#if defined(_MSC_VER)
# pragma once
#endif
#if defined(__GNUC__) && (__GNUC__ > 3 || (__GNUC__ == 3 && __GNUC_MINOR__ > 3))
# pragma once
#endif

#ifndef rt_logging_h
#define rt_logging_h

#include <stddef.h>                     /* size_t */
#include "rtwtypes.h"
#include "rt_mxclassid.h"
#include "rtw_matlogging.h"

#ifndef TMW_NAME_LENGTH_MAX
#define TMW_NAME_LENGTH_MAX 64
#endif
#define mxMAXNAM  TMW_NAME_LENGTH_MAX	/* maximum name length */

/*=========*
 * Defines *
 *=========*/

/*
 * Logging related functions and data structures
 */
typedef double MatReal;                /* "real" data type used in model.mat  */
typedef struct LogVar_Tag LogVar;
typedef struct StructLogVar_Tag StructLogVar;

typedef struct MatrixData_Tag {
  char_T         name[mxMAXNAM];     /* Name of the variable                  */
  int_T          nRows;              /* number of rows                        */
  int_T          nCols;              /* number of columns                     */
  int_T          nDims;              /* number of dimensions                  */
  int_T          _dims[2];           /* most cases, dimensions are 2          */
  int_T          *dims;              /* dimensions of the log variable we
                                        write to at each simulation time step.
                                        E.g: (1) Non-frame data -
                                                 Signal dimension = [2 X 3]
                                                 numDims = 2
                                                 dims[0] = 2, dims[1] = 3
                                             (2) Frame data -
                                                 Signal dimension = [2 X 3]
                                                 numDims = 1
                                                 dims[0] = 3                  */
  void           *re;                /* pointer to real part of the data      */
  void           *im;                /* pointer to imaginary part, if complex */
  DTypeId        dTypeID;            /* data type id                          */
  size_t         elSize;             /* element size in bytes                 */

  RTWLogDataTypeConvert dataTypeConvertInfo;

  mxClassID      mxID;               /* mxId corresponding to this dTypeID    */
  uint32_T       logical;            /* is this a logical array ?             */
  uint32_T       complex;            /* is this a complex matrix?             */
  uint32_T       frameData;          /* is this data frame based?             */
  uint32_T       frameSize;          /* is this data frame based?             */
} MatrixData;

typedef struct ValDimsData_Tag {
  char_T         name[mxMAXNAM];     /* Name of the variable                  */
  int_T          nRows;              /* number of rows                        */
  int_T          nCols;              /* number of columns                     */
  void           **currSigDims;      /* dimensions of current output          */
  int_T          *currSigDimsSize;   /* size in bytes of current sig dims     */
  real_T         *dimsData;          /* pointer to the value of dimension     */
} ValDimsData;

struct LogVar_Tag {
    MatrixData  data;                 /* Container for name, data etc.,       */
    ValDimsData *valDims;             /* field of valueDimensions
                                       1. If all logging signals are fixed-size,
                                          then we set this field to NULL;
                                       2. If any logging signal is variable-size,
                                          then this field will be needed:
                                         1) For fixed-size signal, this field is
                                            an empty matrix;
                                         2) Otherwise, it contains the dimension
                                            information of the logging signal.
                                      */
    int_T      rowIdx;                /* current row index                    */
    int_T      wrapped;               /* number of times the circular buffer
                                       * has wrapped around                   */
    int_T     nDataPoints;            /* total number of data points logged   */
    int_T     usingDefaultBufSize;    /* used to print a message at end       */
    int_T     okayToRealloc;          /* reallocate during sim?               */
    int_T     decimation;             /* decimation factor                    */
    int_T     numHits;                /* decimation hit count                 */

    int_T     *coords;
    int_T     *strides;
    int_T     *currStrides;           /* coords, strides and currStrides will be
                                         needed when logging variable-size
                                         signal to calculate whether the
                                         currently logging value is in the range.
                                         If the current signal is fixed-size,
                                         these pointers will be set to NULLs;
                                         otherwise, we allocate memory for them.
                                         (the size will be nDims in this case)
                                      */

    LogVar    *next;
};

typedef struct SignalsStruct_Tag {
    int_T        numActiveFields;   /* number of active fields                */
    const char_T *fieldNames;
    int_T        numSignals;
    LogVar       *values;
    MatrixData   *dimensions;
    MatrixData   *labels;
    MatrixData   *plotStyles;
    MatrixData   *titles;
    MatrixData   *blockNames;
    MatrixData   *stateNames;
    MatrixData   *crossMdlRef;

    boolean_T    logValueDimensions; /* If there's any variable-size signal
                                         we also should log 'valueDimensions' field
                                      */
    boolean_T    *isVarDims; /* is this signal a variable-size signal? */
} SignalsStruct;

struct StructLogVar_Tag {
    char_T        name[mxMAXNAM];   /* Name of the ML Struct variable         */
    int_T         numActiveFields;  /* number of active fields                */
    boolean_T     logTime;
    void          *time;
    SignalsStruct signals;
    MatrixData    *blockName;

    StructLogVar  *next;
};

#define matUNKNOWN                  0
#define	matINT8                     1
#define	matUINT8                    2
#define	matINT16                    3
#define	matUINT16                   4
#define	matINT32                    5
#define	matUINT32                   6
#define	matFLOAT                    7
#define	matDOUBLE                   9
#define matINT64                   12
#define matUINT64                  13
#define	matMATRIX                  14

/* status of logging "valueDimensions" field */
/*
  NO_LOGVALDIMS:
                 No need to log valueDimensions:
                 All signals are fixed-sized.

  LOGVALDIMS_EMPTYMX:
                 Signals with mixed dimension modes,
                 and the signal logged currently
                 is fixed-sized. So set valueDimensions
                 field to an empty matrix.

  LOGVALDIMS_VARDIMS:
                 Signal logged currently is variable-sized.
*/
typedef enum {
    NO_LOGVALDIMS,
    LOGVALDIMS_EMPTYMX,
    LOGVALDIMS_VARDIMS
} LogValDimsStat;

#ifdef __cplusplus
extern "C" {
#endif

extern mxClassID rt_GetMxIdFromDTypeIdForRSim(BuiltInDTypeId dTypeID);

#ifdef __cplusplus
}
#endif

#ifdef __cplusplus
extern "C" {
#endif

extern mxClassID rt_GetMxIdFromDTypeId(BuiltInDTypeId dTypeID);

#ifdef __cplusplus
}
#endif

#ifdef __cplusplus
extern "C" {
#endif

extern LogVar *rt_CreateLogVarWithConvert(
    RTWLogInfo        *li,
    const real_T      startTime,
    const real_T      finalTime,
    const real_T      inStepSize,
    const char_T      **errStatus,
    const char_T      *varName,
    BuiltInDTypeId    inpDataTypeID,
    const RTWLogDataTypeConvert *pDataTypeConvertInfo,
    int_T             logical,
    int_T             complex,
    int_T             frameData,
    int_T             nCols,
    int_T             nDims,
    const int_T       *dims,
    LogValDimsStat    logValDimsStat,
    void              **currSigDims,
    int_T             *currSigDimsSize,
    int_T             maxRows,
    int_T             decimation,
    real_T            sampleTime,
    int_T             appanedToLogVarsList);

#ifdef __cplusplus
}
#endif

#ifdef __cplusplus
extern "C" {
#endif

extern LogVar *rt_CreateLogVar(RTWLogInfo        *li,
                               const real_T      startTime,
                               const real_T      finalTime,
                               const real_T      inStepSize,
                               const char_T      **errStatus,
                               const char_T      *varName,
                               BuiltInDTypeId    inpDataTypeID,
                               int_T             logical,
                               int_T             complex,
                               int_T             frameData,
                               int_T             nCols,
                               int_T             nDims,
                               const int_T       *dims,
                               LogValDimsStat    logValDimsStat,
                               void              **currSigDims,
                               int_T             *currSigDimsSize,
                               int_T             maxRows,
                               int_T             decimation,
                               real_T            sampleTime,
                               int_T             appanedToLogVarsList);

#ifdef __cplusplus
}
#endif

#ifdef __cplusplus
extern "C" {
#endif

extern StructLogVar *rt_CreateStructLogVar(RTWLogInfo              *li,
                                           const real_T            startTime,
                                           const real_T            finalTime,
                                           const real_T            inStepSize,
                                           const char_T            **errStatus,
                                           const char_T            *varName,
                                           boolean_T               logTime,
                                           int_T                   maxRows,
                                           int_T                   decimation,
                                           real_T                  sampleTime,
                                           const RTWLogSignalInfo  *sigInfo,
                                           const char_T            *blockName);

#ifdef __cplusplus
}
#endif

#ifdef __cplusplus
extern "C" {
#endif

extern const char_T *rt_StartDataLoggingWithStartTime(RTWLogInfo   *li,
                                               const real_T startTime,
                                               const real_T finalTime,
                                               const real_T stepSize,
                                               const char_T **errStatus);

#ifdef __cplusplus
}
#endif

#ifdef __cplusplus
extern "C" {
#endif

#if MAT_FILE == 1

extern const char_T *rt_StartDataLogging(RTWLogInfo   *li,
                                         const real_T finalTime,
                                         const real_T stepSize,
                                         const char_T **errStatus);

#else
#define rt_StartDataLogging(li, finalTime, stepSize, errStatus) NULL /* do nothing */
#endif

#ifdef __cplusplus
}
#endif

#ifdef __cplusplus
extern "C" {
#endif

extern void rt_UpdateLogVar(LogVar *var, const void *data, boolean_T isVarDims);

#ifdef __cplusplus
}
#endif

#ifdef __cplusplus
extern "C" {
#endif

extern void rt_UpdateStructLogVar(StructLogVar *var, const real_T *t, const void *data);

#ifdef __cplusplus
}
#endif

#ifdef __cplusplus
extern "C" {
#endif

#if MAT_FILE == 1

extern const char_T *rt_UpdateTXYLogVars(RTWLogInfo *li, time_T *tPtr);

#else
#define rt_UpdateTXYLogVars(li, tPtr) NULL /* do nothing */
#endif

#ifdef __cplusplus
}
#endif

#ifdef __cplusplus
extern "C" {
#endif

#if MAT_FILE == 1

extern void rt_UpdateSigLogVars(RTWLogInfo *li, time_T *tPtr);

#else
#define rt_UpdateSigLogVars(li, tPtr); /* do nothing */
#endif

#ifdef __cplusplus
}
#endif

#ifdef __cplusplus
extern "C" {
#endif

extern void rt_StopDataLoggingForRaccel(const char_T *file, RTWLogInfo *li, int verbose);

#ifdef __cplusplus
}
#endif

#ifdef __cplusplus
extern "C" {
#endif

#if MAT_FILE == 1

extern void rt_StopDataLogging(const char_T *file, RTWLogInfo *li);

#else
#define rt_StopDataLogging(file, li); /* do nothing */
#endif

#ifdef __cplusplus
}
#endif

#endif /* rt_logging_h */
```

### rt_logging_mmi.h
```c
/* $Revision: 1.1.6.5 $
 *
 * Copyright 1994-2004 The MathWorks, Inc.
 *
 * File: rt_logging_mmi.h
 *
 * Abstract:
 */

#ifndef rt_logging_mmi_h
#define rt_logging__mmi_h

#include <stdlib.h>
#include "rtwtypes.h"
#include "rtw_matlogging.h"
#include "rtw_modelmap.h"

#ifdef __cplusplus
extern "C" {
#endif

const char_T * rt_FillStateSigInfoFromMMI(RTWLogInfo   *li,
                                          const char_T **errStatus);

void rt_CleanUpForStateLogWithMMI(RTWLogInfo *li);

const char_T * rt_FillSigLogInfoFromMMI(RTWLogInfo    *li,
                                        const char_T  **errStatus);

void rt_CleanUpForSigLogWithMMI(RTWLogInfo *li);

#ifdef __cplusplus
}
#endif

#endif /*  rt_logging_h */
```

### rt_math.h
```c
/* Copyright 2010 The MathWorks, Inc. */
#ifndef RTW_HEADER_rt_math_h_
#define RTW_HEADER_rt_math_h_

#define rt_MAXf_snf(a, b)              (( ((a) >= (b)) || rtIsNaNF(b) ) ? (a) : (b))
#define rt_MAXd_snf(a, b)              (( ((a) >= (b)) || rtIsNaN(b) ) ? (a) : (b))
#define rt_MAXf(a, b)                  (((a) >= (b)) ? (a) : (b))
#define rt_MAXd(a, b)                  (((a) >= (b)) ? (a) : (b))
#define rt_MAX(a, b)                   (((a) >= (b)) ? (a) : (b))

#define rt_MINf_snf(a, b)              (( ((a) <= (b)) || rtIsNaNF(b) ) ? (a) : (b))
#define rt_MINd_snf(a, b)              (( ((a) <= (b)) || rtIsNaN(b) ) ? (a) : (b))
#define rt_MINf(a, b)                  (((a) <= (b)) ? (a) : (b))
#define rt_MINd(a, b)                  (((a) <= (b)) ? (a) : (b))
#define rt_MIN(a, b)                   (((a) <= (b)) ? (a) : (b))

#define rt_SIGNf_snf(a)                ( ((a) < 0.0F) ? -1.0F : ((a) > 0.0F) ? 1.0F : ((a) == 0.0F) ? 0.0F : (rtNaNF) )
#define rt_SIGNd_snf(a)                ( ((a) < 0.0) ? -1.0 : ((a) > 0.0) ? 1.0 : ((a) == 0.0) ? 0.0 : (rtNaN) )
#define rt_SIGNf(a)                    ( ((a) < 0.0F) ? -1.0F : ((a) > 0.0F) ? 1.0F : 0.0F )
#define rt_SIGNd(a)                    ( ((a) < 0.0) ? -1.0 : ((a) > 0.0) ? 1.0 : 0.0 )
#define rt_SGN(a)                      ( ((a) < 0) ? -1 : ((a) > 0) ? 1 : 0 )
#define rt_UNSGN(a)                    ( ((a) > 0U) ? 1U : 0U )

#define rt_SATURATE(sig,ll,ul)         (((sig) >= (ul)) ? (ul) : (((sig) <= (ll)) ? (ll) : (sig)) )

#define rt_ABS(a)                      ( ((a) >= 0) ? (a) : -(a) )

#endif                                 /* RTW_HEADER_rt_math_h_ */
```

### rt_matrixlib.h
```c
#ifndef rt_matrixlib_h
#define rt_matrixlib_h

/* Copyright 2007-2010 The MathWorks, Inc.
 *
 * File    : rt_matrixlib.h
 * Abstract:
 *     Function prototypes for .c sources in rtw/c/src/matrixmath.
 *
 */

/* $Revision: 1.1.6.2 $ */

/*==========*
 * Includes *
 *==========*/

#include "rtwtypes.h"
#include <limits.h>

#ifdef __cplusplus
extern "C" {
#endif

/* Matrix Multiplication Utility Functions */
extern void rt_MatMultRR_Dbl(real_T         *y,
                             const real_T   *A,
                             const real_T   *B,
                             const int_T dims[3]);

#ifdef CREAL_T
extern void rt_MatMultRC_Dbl(creal_T       *y,
                             const real_T  *A,
                             const creal_T *B,
                             const int_T dims[3]);

extern void rt_MatMultCR_Dbl(creal_T       *y,
                             const creal_T *A,
                             const real_T  *B,
                             const int_T dims[3]);

extern void rt_MatMultCC_Dbl(creal_T       *y,
                             const creal_T *A,
                             const creal_T *B,
                             const int_T dims[3]);
#endif

extern void rt_MatMultRR_Sgl(real32_T       *y,
                             const real32_T *A,
                             const real32_T *B,
                             const int_T  dims[3]);

#ifdef CREAL_T
extern void rt_MatMultRC_Sgl(creal32_T       *y,
                             const real32_T  *A,
                             const creal32_T *B,
                             const int_T   dims[3]);

extern void rt_MatMultCR_Sgl(creal32_T       *y,
                             const creal32_T *A,
                             const real32_T  *B,
                             const int_T   dims[3]);

extern void rt_MatMultCC_Sgl(creal32_T       *y,
                             const creal32_T *A,
                             const creal32_T *B,
                             const int_T   dims[3]);
#endif

extern void rt_MatMultAndIncRR_Dbl(real_T       *y,
                                   const real_T *A,
                                   const real_T *B,
                                   const int_T dims[3]);

#ifdef CREAL_T
extern void rt_MatMultAndIncRC_Dbl(creal_T       *y,
                                   const real_T  *A,
                                   const creal_T *B,
                                   const int_T dims[3]);

extern void rt_MatMultAndIncCR_Dbl(creal_T       *y,
                                   const creal_T *A,
                                   const real_T  *B,
                                   const int_T dims[3]);

extern void rt_MatMultAndIncCC_Dbl(creal_T       *y,
                                   const creal_T *A,
                                   const creal_T *B,
                                   const int_T dims[3]);
#endif
extern void rt_MatMultAndIncRR_Sgl(real32_T       *y,
                                   const real32_T *A,
                                   const real32_T *B,
                                   const int_T  dims[3]);

#ifdef CREAL_T
extern void rt_MatMultAndIncRC_Sgl(creal32_T       *y,
                                   const real32_T  *A,
                                   const creal32_T *B,
                                   const int_T   dims[3]);

extern void rt_MatMultAndIncCR_Sgl(creal32_T       *y,
                                   const creal32_T *A,
                                   const real32_T  *B,
                                   const int_T   dims[3]);

extern void rt_MatMultAndIncCC_Sgl(creal32_T       *y,
                                   const creal32_T *A,
                                   const creal32_T *B,
                                   const int_T   dims[3]);
#endif

/* Matrix Inversion Utility Functions */
extern void rt_lu_real(real_T      *A,
                       const int_T n,
                       int32_T     *piv);

#ifdef CREAL_T
extern void rt_lu_cplx(creal_T *A,
                       const int_T n,
                       int32_T *piv);
#endif

extern void rt_lu_real_sgl(real32_T      *A,
                           const int_T n,
                           int32_T     *piv);

#ifdef CREAL_T
extern void rt_lu_cplx_sgl(creal32_T *A,
                           const int_T n,
                           int32_T *piv);
#endif

extern void rt_BackwardSubstitutionRR_Dbl(real_T          *pU,
                                          const real_T    *pb,
                                          real_T          *x,
                                          int_T            N,
                                          int_T            P,
                                          boolean_T        unit_upper);

#ifdef CREAL_T
extern void rt_BackwardSubstitutionRC_Dbl(real_T          *pU,
                                          const creal_T   *pb,
                                          creal_T         *x,
                                          int_T            N,
                                          int_T            P,
                                          boolean_T        unit_upper);

extern void rt_BackwardSubstitutionCC_Dbl(creal_T         *pU,
                                          const creal_T   *pb,
                                          creal_T         *x,
                                          int_T            N,
                                          int_T            P,
                                          boolean_T        unit_upper);
#endif

extern void rt_ForwardSubstitutionRR_Dbl(real_T        *pL,
                                         const real_T  *pb,
                                         real_T        *x,
                                         int_T          N,
                                         int_T          P,
                                         const int32_T *piv,
                                         boolean_T      unit_lower);

#ifdef CREAL_T
extern void rt_ForwardSubstitutionRC_Dbl(real_T        *pL,
                                         const creal_T   *pb,
                                         creal_T   *x,
                                         int_T     N,
                                         int_T     P,
                                         const int32_T   *piv,
                                         boolean_T unit_lower);

extern void rt_ForwardSubstitutionCR_Dbl(creal_T   *pL,
                                         const real_T    *pb,
                                         creal_T   *x,
                                         int_T     N,
                                         int_T     P,
                                         const int32_T   *piv,
                                         boolean_T unit_lower);

extern void rt_ForwardSubstitutionCC_Dbl(creal_T   *pL,
                                         const creal_T   *pb,
                                         creal_T   *x,
                                         int_T     N,
                                         int_T     P,
                                         const int32_T   *piv,
                                         boolean_T unit_lower);
#endif

extern void rt_BackwardSubstitutionRR_Sgl(real32_T          *pU,
                                          const real32_T    *pb,
                                          real32_T          *x,
                                          int_T              N,
                                          int_T              P,
                                          boolean_T          unit_upper);

#ifdef CREAL_T
extern void rt_BackwardSubstitutionRC_Sgl(real32_T          *pU,
                                          const creal32_T   *pb,
                                          creal32_T         *x,
                                          int_T              N,
                                          int_T              P,
                                          boolean_T          unit_upper);

extern void rt_BackwardSubstitutionCC_Sgl(creal32_T         *pU,
                                          const creal32_T   *pb,
                                          creal32_T         *x,
                                          int_T              N,
                                          int_T              P,
                                          boolean_T          unit_upper);
#endif

extern void rt_ForwardSubstitutionRR_Sgl(real32_T    *pL,
                                         const real32_T    *pb,
                                         real32_T    *x,
                                         int_T     N,
                                         int_T     P,
                                         const int32_T   *piv,
                                         boolean_T unit_lower);

#ifdef CREAL_T
extern void rt_ForwardSubstitutionRC_Sgl(real32_T    *pL,
                                         const creal32_T   *pb,
                                         creal32_T   *x,
                                         int_T     N,
                                         int_T     P,
                                         const int32_T   *piv,
                                         boolean_T unit_lower);

extern void rt_ForwardSubstitutionCR_Sgl(creal32_T   *pL,
                                         const real32_T    *pb,
                                         creal32_T   *x,
                                         int_T     N,
                                         int_T     P,
                                         const int32_T   *piv,
                                         boolean_T unit_lower);

extern void rt_ForwardSubstitutionCC_Sgl(creal32_T   *pL,
                                         const creal32_T   *pb,
                                         creal32_T   *x,
                                         int_T     N,
                                         int_T     P,
                                         const int32_T   *piv,
                                         boolean_T unit_lower);
#endif

extern void rt_MatDivRR_Dbl(real_T        *Out,
                            const real_T  *In1,
                            const real_T  *In2,
                            real_T        *lu,
                            int32_T       *piv,
                            real_T        *x,
                            const int_T    dims[3]);

#ifdef CREAL_T
extern void rt_MatDivRC_Dbl(creal_T       *Out,
                            const real_T  *In1,
                            const creal_T *In2,
                            real_T        *lu,
                            int32_T       *piv,
                            creal_T       *x,
                            const int_T    dims[3]);

extern void rt_MatDivCR_Dbl(creal_T       *Out,
                            const creal_T *In1,
                            const real_T  *In2,
                            creal_T       *lu,
                            int32_T       *piv,
                            creal_T       *x,
                            const int_T    dims[3]);

extern void rt_MatDivCC_Dbl(creal_T       *Out,
                            const creal_T *In1,
                            const creal_T *In2,
                            creal_T       *lu,
                            int32_T       *piv,
                            creal_T       *x,
                            const int_T    dims[3]);
#endif

extern void rt_MatDivRR_Sgl(real32_T        *Out,
                            const real32_T  *In1,
                            const real32_T  *In2,
                            real32_T        *lu,
                            int32_T         *piv,
                            real32_T        *x,
                            const int_T      dims[3]);

#ifdef CREAL_T
extern void rt_MatDivRC_Sgl(creal32_T       *Out,
                            const real32_T  *In1,
                            const creal32_T *In2,
                            real32_T        *lu,
                            int32_T         *piv,
                            creal32_T       *x,
                            const int_T      dims[3]);

extern void rt_MatDivCR_Sgl(creal32_T       *Out,
                            const creal32_T *In1,
                            const real32_T  *In2,
                            creal32_T       *lu,
                            int32_T         *piv,
                            creal32_T       *x,
                            const int_T      dims[3]);

extern void rt_MatDivCC_Sgl(creal32_T       *Out,
                            const creal32_T *In1,
                            const creal32_T *In2,
                            creal32_T       *lu,
                            int32_T         *piv,
                            creal32_T       *x,
                            const int_T      dims[3]);
#endif

/* Matrix multiplication defines */

/* Quick (approximate) complex absolute value: */
#define CQABS(X) (fabs((X).re) + fabs((X).im))

/* Quick (approximate) complex absolute value for singles: */
#define CQABSSGL(X) (real32_T)(fabs( (real_T) (X).re) + fabs( (real_T) (X).im))

#ifdef CREAL_T
extern void rt_ComplexTimes_Dbl(creal_T       *Out,
                                const creal_T In1,
                                const creal_T In2);

extern void rt_ComplexRDivide_Dbl(creal_T       *Out,
                                  const creal_T In1,
                                  const creal_T In2);

extern void rt_ComplexReciprocal_Dbl(creal_T       *Out,
                                     const creal_T In1);

extern void rt_ComplexTimes_Sgl(creal32_T       *Out,
                                const creal32_T In1,
                                const creal32_T In2);

extern void rt_ComplexRDivide_Sgl(creal32_T       *Out,
                                  const creal32_T In1,
                                  const creal32_T In2);

extern void rt_ComplexReciprocal_Sgl(creal32_T       *Out,
                                     const creal32_T In1);

#endif

extern real_T rt_Hypot_Dbl(real_T In1,
                           real_T In2);

extern real32_T rt_Hypot_Sgl(real32_T In1,
                             real32_T In2);

#ifdef __cplusplus
}
#endif

#endif /* rt_matrixlib_h */
```

### rt_matrx.h
```c
/*
 * @(#)rt_matrx.h    generated by: makeheader 5.1.5  Tue May 24 21:25:56 2011
 *
 *		built from:	rt_matrx.c
 */

#if defined(_MSC_VER)
# pragma once
#endif
#if defined(__GNUC__) && (__GNUC__ > 3 || (__GNUC__ == 3 && __GNUC_MINOR__ > 3))
# pragma once
#endif

#ifndef rt_matrx_h
#define rt_matrx_h

/*
 * Copyright 1994-2010 The MathWorks, Inc.
 * $Revision: 1.1.6.7 $
 * $Date: 2010/09/13 14:17:56 $
 */

/*==========*
 * Includes *
 *==========*/

#if defined(MATLAB_MEX_FILE)
# error "rt_matrix cannot be used within a mex file. It is for codegen only."
#endif

#include <stdlib.h>    /* needed for malloc, calloc, free, realloc */
#include <string.h>    /* needed for strlen                        */
#include "rtwtypes.h"  /* needed for real_T                        */
#include "rt_mxclassid.h" /* needed for mxClassID                     */

/*==========*
 * Typedefs *
 *==========*/

#ifndef rt_typedefs_h
#define rt_typedefs_h

#if !defined(TYPEDEF_MX_ARRAY)
# define TYPEDEF_MX_ARRAY
  typedef real_T mxArray;
#endif

typedef real_T mxChar;

#if !defined(TMW_NAME_LENGTH_MAX)
#define TMW_NAME_LENGTH_MAX 64
#endif
#define mxMAXNAM  TMW_NAME_LENGTH_MAX	/* maximum name length */

typedef enum {
    mxREAL,
    mxCOMPLEX
} mxComplexity;

#endif /* rt_typedefs_h */

/*==================*
 * Extern variables *
 *==================*/

#ifdef __cplusplus
extern "C" {
#endif

extern real_T rtInf;
extern real_T rtMinusInf;
extern real_T rtNaN;

#ifdef __cplusplus
}
#endif

/*=======================================*
 * Defines for mx Routines and constants *
 *=======================================*/

#define mxCalloc(n,size) \
        calloc(n,size)

#define mxCreateCharArray(ndim, dims) \
        mxCreateNumericArray(ndim, dims, mxCHAR_CLASS);

#define mxDestroyArray(pa) \
        if (pa) free(pa)

/* NOTE: You cannot mxFree(mxGetPr(pa)) !!! */
#define mxFree(ptr) \
        if(ptr)free(ptr)

#define mxGetClassID(pa) \
        mxDOUBLE_CLASS

/* NOTE: mxGetClassName(pa) returns "double" even on a character array */
#define mxGetClassName(pa) \
        "double"

#define mxGetData(pa) \
        ((void *)(&((pa)[2])))

#define mxGetElementSize(pa) \
        (sizeof(real_T))

#define mxGetInf() \
        rtInf

#define mxGetM(pa) \
        ((size_t) ((pa)[0]))
#define mxGetN(pa) \
        ((size_t) ((pa)[1]))

#define mxGetNaN() \
        rtNaN

#define mxGetNumberOfDimensions(pa) \
        (2)
#define mxGetNumberOfElements(pa) \
        (mxGetM(pa)*mxGetN(pa))

/* NOTE: mxGetPr() of an empty matrix does NOT return NULL */
#define mxGetPr(pa) \
        ( &((pa)[2]) )

#define mxGetScalar(pa) \
        ((pa)[2])

#define mxIsComplex(pa) \
        false

#define mxIsDouble(pa) \
        true

#define mxIsEmpty(pa) \
        (mxGetM(pa)==0 || mxGetN(pa)==0)

#define mxIsFinite(r) \
        ((r)>rtMinusInf && (r)<rtInf)

#define mxIsInf(r) \
        ((r)==rtInf || (r)==rtMinusInf)

#define mxIsInt16(pa) \
        false

#define mxIsInt32(pa) \
        false

#define mxIsInt8(pa) \
        false

#define mxIsLogical(pa) \
        false

#define mxIsNumeric(pa) \
        true

#define mxIsSingle(pa) \
        false

#define mxIsSparse(pa) \
        false

#define mxIsStruct(pa) \
        false

#define mxIsUint16(pa) \
        false

#define mxIsUint32(pa) \
        false

#define mxIsUint8(pa) \
        false

#define mxMalloc(n) \
        malloc(n)

#define mxRealloc(p,n) \
        realloc(p,n)

/*==========================*
 * Visible/extern functions *
 *=========================*/

#ifdef __cplusplus
extern "C" {
#endif

extern mxArray *rt_mxCreateCharMatrixFromStrings(int_T m, const char_T **str);

#ifdef __cplusplus
}
#endif

#ifdef __cplusplus
extern "C" {
#endif

extern mxArray *rt_mxCreateString(const char *str);

#ifdef __cplusplus
}
#endif

#ifdef __cplusplus
extern "C" {
#endif

extern mxArray *rt_mxCreateDoubleMatrix(int m, int n, mxComplexity flag);

#ifdef __cplusplus
}
#endif

#ifdef __cplusplus
extern "C" {
#endif

extern mxArray *rt_mxCreateNumericArray(int_T ndims, const int_T *dims,
                                        mxClassID classid, mxComplexity flag);

#ifdef __cplusplus
}
#endif

#ifdef __cplusplus
extern "C" {
#endif

extern mxArray *rt_mxDuplicateArray(const mxArray *pa);

#ifdef __cplusplus
}
#endif

#ifdef __cplusplus
extern "C" {
#endif

extern const int_T *rt_mxGetDimensions(const mxArray *pa);

#ifdef __cplusplus
}
#endif

#ifdef __cplusplus
extern "C" {
#endif

extern real_T rt_mxGetEps(void);

#ifdef __cplusplus
}
#endif

#ifdef __cplusplus
extern "C" {
#endif

extern int_T rt_mxGetString(const mxArray *pa, char_T *buf, int_T buflen);

#ifdef __cplusplus
}
#endif

#define mxCreateCharMatrixFromStrings(m, str) \
        rt_mxCreateCharMatrixFromStrings(m, str)

#define mxCreateString(str) \
        rt_mxCreateString(str)

#define mxCreateDoubleMatrix(m, n, flag) \
        rt_mxCreateDoubleMatrix(m, n, flag)

#define mxCreateNumericArray(ndims, dims, classid, flag) \
        rt_mxCreateNumericArray(ndims, dims, classid, flag)

#define mxDuplicateArray(pa) \
        rt_mxDuplicateArray(pa)

#define mxGetDimensions(pa) \
        rt_mxGetDimensions(pa)

#define mxGetEps() \
        rt_mxGetEps()

#define mxGetString(pa, buf, buflen) \
        rt_mxGetString(pa, buf, buflen)

/*=========================*
 * Unsupported mx Routines *
 *=========================*/

#define mxCalcSingleSubscript(pa,nsubs,subs) \
        mxCalcSingleSubscript_is_not_supported_in_Simulink_Coder

#define mxCreateCellArray(ndim,dims) \
        mxCreateCellArray_is_not_supported_in_Simulink_Coder

#define mxCreateCellMatrix(m,n) \
        mxCreateCellMatrix_is_not_supported_in_Simulink_Coder

#define mxCreateSparse(pm,pn,pnzmax,pcmplx_flg) \
        mxCreateSparse_is_not_supported_in_Simulink_Coder

#define mxCreateStructArray(ndim,dims,nfields,fieldnames) \
        mxCreateStructArray_is_not_supported_in_Simulink_Coder

#define mxCreateStructMatrix(m,n,nfields,fieldnames) \
        mxCreateStructMatrix_is_not_supported_in_Simulink_Coder

#define mxGetCell(pa,i) \
        mxGetCell_is_not_supported_in_Simulink_Coder

#define mxGetField(pa,i,fieldname) \
        mxGetField_is_not_supported_in_Simulink_Coder

#define mxGetFieldByNumber(s,i,fieldnum) \
        mxGetFieldByNumber_is_not_supported_in_Simulink_Coder

#define mxGetFieldNameByNumber(pa,n) \
        mxGetFieldNameByNumber_is_not_supported_in_Simulink_Coder

#define mxGetFieldNumber(pa,fieldname) \
        mxGetFieldNumber_is_not_supported_in_Simulink_Coder

#define mxGetImagData(pa) \
        mxGetImagData_is_not_supported_in_Simulink_Coder

#define mxGetIr(ppa) \
        mxGetIr_is_not_supported_in_Simulink_Coder

#define mxGetJc(ppa) \
        mxGetJc_is_not_supported_in_Simulink_Coder

#define mxGetNumberOfFields(pa) \
        mxGetNumberOfFields_is_not_supported_in_Simulink_Coder

#define mxGetNzmax(pa) \
        mxGetNzmax_is_not_supported_in_Simulink_Coder

#define mxGetPi(pa) \
        mxGetPi_is_not_supported_in_Simulink_Coder

#define mxIsFromGlobalWS(pa) \
        mxIsFromGlobalWS_is_not_supported_in_Simulink_Coder

#define mxIsNaN(r) \
        mxIsNaN_is_not_supported_in_Simulink_Coder

#define mxIsChar(pa) \
        mxIsChar_is_not_supported_in_Simulink_Coder

#define mxIsClass(pa,class) \
        mxIsClass_is_not_supported_in_Simulink_Coder

#define mxIsCell(pa) \
        mxIsCell_is_not_supported_in_Simulink_Coder

#define mxSetCell(pa,i,value) \
        mxSetCell_is_not_supported_in_Simulink_Coder

#define mxSetClassName(pa,classname) \
        mxSetClassName_is_not_supported_in_Simulink_Coder

#define mxSetData(pa,pr) \
        mxSetData_is_not_supported_in_Simulink_Coder

#define mxSetDimensions(pa, size, ndims) \
        mxSetDimensions_is_not_supported_in_Simulink_Coder

#define mxSetField(pa,i,fieldname,value) \
        mxSetField_is_not_supported_in_Simulink_Coder

#define mxSetFieldByNumber(pa, index, fieldnum, value) \
        mxSetFieldByNumber_is_not_supported_in_Simulink_Coder

#define mxSetFromGlobalWS(pa,global) \
        mxSetFromGlobalWS_is_not_supported_in_Simulink_Coder

#define mxSetImagData(pa,pv) \
        mxSetImagData_is_not_supported_in_Simulink_Coder

#define mxSetIr(ppa,ir) \
        mxSetIr_is_not_supported_in_Simulink_Coder

#define mxSetJc(ppa,jc) \
        mxSetJc_is_not_supported_in_Simulink_Coder

#define mxSetM(pa, m) \
        mxSetM_is_not_supported_in_Simulink_Coder

#define mxSetN(pa, m) \
        mxSetN_is_not_supported_in_Simulink_Coder

#define mxSetPr(pa,pr) \
        mxSetPr_is_not_supported_in_Simulink_Coder

#define mxSetNzmax(pa,nzmax) \
        mxSetNzmax_is_not_supported_in_Simulink_Coder

#define mxSetPi(pa,pv) \
        mxSetPi_is_not_supported_in_Simulink_Coder

/*==========================*
 * Unsupported mex routines *
 *==========================*/

#define mexPrintAssertion(test,fname,linenum,message) \
        mexPrintAssertion_is_not_supported_by_Simulink_Coder

#define mexEvalString(str) \
        mexEvalString_is_not_supported_by_Simulink_Coder

#define mexErrMsgTxt(str) \
        mexErrMsgTxt_is_not_supported_by_Simulink_Coder

#define mexWarnMsgTxt(warning_msg) \
        mexWarnMsgTxt_is_not_supported_by_Simulink_Coder

#define mexPrintf \
        mexPrintf_is_not_supported_by_Simulink_Coder

#define mexMakeArrayPersistent(pa) \
        mexMakeArrayPersistent_is_not_supported_by_Simulink_Coder

#define mexMakeMemoryPersistent(ptr) \
        mexMakeMemoryPersistent_is_not_supported_by_Simulink_Coder

#define mexLock() \
        mexLock_is_not_supported_by_Simulink_Coder

#define mexUnlock() \
        mexUnlock_is_not_supported_by_Simulink_Coder

#define mexFunctionName() \
        mexFunctionName_is_not_supported_by_Simulink_Coder

#define mexIsLocked() \
        mexIsLocked_is_not_supported_by_Simulink_Coder

#define mexGetFunctionHandle() \
        mexGetFunctionHandle_is_not_supported_by_Simulink_Coder

#define mexCallMATLABFunction() \
        mexCallMATLABFunction_is_not_supported_by_Simulink_Coder

#define mexRegisterFunction() \
        mexRegisterFunction_is_not_supported_by_Simulink_Coder

#define mexSet(handle,property,value) \
        mexSet_is_not_supported_by_Simulink_Coder

#define mexGet(handle,property) \
        mexGet_is_not_supported_by_Simulink_Coder

#define mexCallMATLAB(nlhs,plhs,nrhs,prhs,fcn) \
        mexCallMATLAB_is_not_supported_by_Simulink_Coder

#define mexSetTrapFlag(flag) \
        mexSetTrapFlag_is_not_supported_by_Simulink_Coder

#define mexUnlink(a) \
        mexUnlink_is_not_supported_by_Simulink_Coderw

#define mexSubsAssign(plhs,sub,nsubs,prhs) \
        mexSubsAssign_is_not_supported_by_Simulink_Coder

#define mexSubsReference(prhs,subs,nsubs) \
        mexSubsReference_is_not_supported_by_Simulink_Coder

#define mexPrintAssertion(test,fname,linenum,message) \
        mexPrintAssertion_is_not_supported_by_Simulink_Coder

#define mexAddFlops(count) \
        mexAddFlops_is_not_supported_by_Simulink_Coder

#define mexIsGlobal(pa) \
        mexIsGlobal_is_not_supported_by_Simulink_Coder

#define mexAtExit(fcn) \
        mexAtExit_is_not_supported_by_Simulink_Coder

#endif /* rt_matrx_h */
```

### rt_mxclassid.h
```c
/* Copyright 1994-2004 The MathWorks, Inc.
 *
 * File    : rt_mxclassid.h
 * Abstract:
 *   Definition of enum mxClassID
 *
 */

/* $Revision: 1.1.6.1 $ */

#ifndef __rt_mxclassid_h__
#define __rt_mxclassid_h__

typedef enum {
	mxUNKNOWN_CLASS = 0,
	mxCELL_CLASS = 1,
	mxSTRUCT_CLASS,
	mxLOGICAL_CLASS,
	mxCHAR_CLASS,
	mxRESERVED5_CLASS, /* mxVOID_CLASS */
	mxDOUBLE_CLASS,
	mxSINGLE_CLASS,
	mxINT8_CLASS,
	mxUINT8_CLASS,
	mxINT16_CLASS,
	mxUINT16_CLASS,
	mxINT32_CLASS,
	mxUINT32_CLASS,
	mxINT64_CLASS,		/* place holder - future enhancements */
	mxUINT64_CLASS,		/* place holder - future enhancements */
	mxRESERVED16_CLASS, /* mxFUNCTION_CLASS */
	mxRESERVED17_CLASS, /* mxOPAQUE_CLASS */
	mxOBJECT_CLASS
} mxClassID;

#endif /* __rt_mxclassid_h__ */

/* [EOF] rt_mxclass_id.h */
```

### rt_sim.h
```c
/*
 * Copyright 1994-2009 The MathWorks, Inc.
 *
 * File: rt_sim.h     $Revision: 1.15.4.4 $
 *
 * Abstract:
 *	Function prototypes for routines which perform one time step of
 *	a real-time single tasking or multitasking system.
 */

#ifndef __RT_SIM__
#define __RT_SIM__

#ifdef __cplusplus
extern "C" {
#endif

/*
 * Functions that do not require the SimStruct as an arg
 */
#define rttiSetTaskTime(tPtr,sti,time) (tPtr)[sti]=(time)

#define rttiSetSampleHitInTask(perTaskSampHits,numSampTimes,task_j,task_i,hit) \
    (perTaskSampHits)[(task_j) + ((task_i) * (numSampTimes))] = (hit)

extern const char *rt_SimInitTimingEngine(int_T       rtmNumSampTimes,
                                          real_T      rtmStepSize,
                                          real_T      *rtmSampleTimePtr,
                                          real_T      *rtmOffsetTimePtr,
                                          int_T       *rtmSampleHitPtr,
                                          int_T       *rtmSampleTimeTaskIDPtr,
                                          real_T      rtmTStart,
                                          SimTimeStep *rtmSimTimeStepPtr,
                                          void        **rtmTimingDataPtr);
#ifdef RT_MALLOC
extern void rt_SimDestroyTimingEngine(void *rtmTimingData);
#endif

#if !defined(MULTITASKING)
  extern void  rt_SimUpdateDiscreteTaskSampleHits(int_T  rtmNumSampTimes,
                                                  void   *rtmTimingData,
                                                  int_T  *rtmSampleHitPtr,
                                                  real_T *rtmTPtr);
#  ifndef RT_MALLOC
     extern time_T rt_SimGetNextSampleHit(void);
#  else
     extern time_T rt_SimGetNextSampleHit(void   *rtmTimingData,
                                          int_T rtmNumSampTimes);
#  endif
#else
#  ifndef USE_RTMODEL
     extern time_T rt_SimUpdateDiscreteEvents(int_T  rtmNumSampTimes,
                                              void   *rtmTimingData,
                                              int_T  *rtmSampleHitPtr,
                                              int_T  *rtmPerTaskSampleHits);
#  endif
  extern void   rt_SimUpdateDiscreteTaskTime(real_T *rtmTPtr,
                                             void   *rtmTimingData,
                                             int    tid);
#endif

/*
 * Functions maintained for backwards compatibility
 */
#ifndef USE_RTMODEL
  extern const char *rt_InitTimingEngine(SimStruct *S);
# ifdef RT_MALLOC
    extern void   rt_DestroyTimingEngine(SimStruct *S);
# endif

# if !defined(MULTITASKING)
    extern void   rt_UpdateDiscreteTaskSampleHits(SimStruct *S);
#   ifndef RT_MALLOC
      extern time_T rt_GetNextSampleHit(void);
#   else
      extern time_T rt_GetNextSampleHit(SimStruct *S);
#   endif

# else
    extern time_T rt_UpdateDiscreteEvents(SimStruct *S);
    extern void   rt_UpdateDiscreteTaskTime(SimStruct *S, int tid);
# endif
#endif /* !(USE_RTMODEL) */

#ifdef __cplusplus
}
#endif

#endif /* __RT_SIM__ */
```

### rt_size_check.h
```c
/* Copyright 2009-2010 The MathWorks, Inc. */
#ifndef rt_size_check_h
#define rt_size_check_h

#include "simstruc.h"

void
rtErrorMsgID(SimStruct*  S, const char* msgID);

void
rtSizeEqCheck1D(SimStruct*  S, int  dims1, int dims2);

void
rtSizeEqCheckND(SimStruct*  S, int* dims1, int* dims2, int nDims) ;

#endif
```

### rtiostream.h
```c
/*
 * Copyright 2007-2008 The MathWorks, Inc.
 *
 * File: rtiostream.h     $Revision: 1.1.6.2 $
 *
 * Abstract:
 *  Function prototypes and defines for rtIOStream API.
 */

#ifndef RTIOSTREAM_H
#define RTIOSTREAM_H

#include <stddef.h>

#define RTIOSTREAM_ERROR (-1)
#define RTIOSTREAM_NO_ERROR (0)

/* Note: if the functions declared in this file should be compiled into a shared
 * library (e.g. a .dll file on Windows), you must ensure that the functions are
 * externally visible. The procedure to achieve this depends on the compiler and
 * linker you are using. For example, on Windows, you may need to provide an
 * exports definition .def file that lists all of the functions to be
 * exported; see ./rtiostream/rtiostream_pc.def for a suitable .def file.
 */

int rtIOStreamOpen(
    int    argc,
    void * argv[]
);

int rtIOStreamSend(
    int          streamID,
    const void * src,
    size_t       size,
    size_t     * sizeSent
    );

int rtIOStreamRecv(
    int      streamID,
    void   * dst,
    size_t   size,
    size_t * sizeRecvd
    );

int rtIOStreamClose(
    int streamID
    );

#endif /* #ifndef RTIOSTREAM_H */
```

### rtmcmacros.h
```c
/*
 * Copyright 1994-2002 The MathWorks, Inc.
 *
 * File: rtmcmacros.h     $Revision: 1.1 $
 *
 * Abstract:
 * API glue for calling rt_OneStep.  These macros are used to create
 * a structure with the elements in the rtModel structure that are
 * required to be passed to rt_OneStep.
 */

#ifndef _RTW_HEADER_rtmcmacros_h_
# define _RTW_HEADER_rtmcmacros_h_

/* Real-time Model Common Data Structure */
typedef struct {
  const char            **errorStatus;
  RTWLogInfo            **rtwLogInfo;
  RTWExtModeInfo        **extModeInfo;
  RTWRTModelMethodsInfo *modelMethodsInfo;
  RTWSolverInfo         **solverInfo;
  int_T                  *numSampTimes;
  time_T                **t;
  void                  **timingData;
  SimTimeStep            *simTimeStep;
  int_T                 **sampleHits;
  int_T                 **perTaskSampleHitsPtr;
  boolean_T              *stopRequested;
  time_T                **sampleTimes;
  int_T                 **sampleTimeTaskIDPtr;
} rtModelCommon;

#define rtmcsetCommon(MC, M)                                  \
    MC.errorStatus         = &rtmGetErrorStatus(M);           \
    MC.rtwLogInfo          = &rtmGetRTWLogInfo(M);            \
    MC.extModeInfo         = &rtmGetRTWExtModeInfo(M);        \
    MC.modelMethodsInfo     = &rtmGetRTWRTModelMethodsInfo(M); \
    MC.solverInfo           = &rtmGetRTWSolverInfo(M);         \
    MC.numSampTimes         = &rtmGetNumSampleTimes(M);        \
    MC.t                    = &rtmGetTPtr(M);                  \
    MC.timingData           = &rtmGetTimingData(M);            \
    MC.simTimeStep          = &rtmGetSimTimeStep(M);           \
    MC.sampleHits           = &rtmGetSampleHitPtr(M);          \
    MC.perTaskSampleHitsPtr = &rtmGetPerTaskSampleHitsPtr(M);  \
    MC.stopRequested        = &rtmGetStopRequested(M);         \
    MC.sampleTimes          = &rtmGetSampleTimePtr(M);         \
    MC.sampleTimeTaskIDPtr  = &rtmGetSampleTimeTaskIDPtr(M);

# define rtmcGetErrorStatus(rtmc)   (*rtmc->errorStatus)
# define rtmcGetRTWLogInfo(rtmc)   (*rtmc->rtwLogInfo)
# define rtmcGetRTWExtModeInfo(rtmc) (*rtmc->extModeInfo)
# define rtmcGetRTWRTModelMethodsInfo(rtmc) (*rtmc->modelMethodsInfo)
# define rtmcGetRTWSolverInfo(rtmc) (*rtmc->solverInfo)
# define rtmcGetNumSampleTimes(rtmc) (*rtmc->numSampTimes)
# define rtmcGetTPtr(rtmc) (*rtmc->t)
# define rtmcGetTimingData(rtmc) (*rtmc->timingData)
# define rtmcGetSimTimeStep(rtmc) (*rtmc->simTimeStep)
# define rtmcGetSampleHitPtr(rtmc) (*rtmc->sampleHits)
# define rtmcGetPerTaskSampleHitsPtr(rtmc) (*rtmc->perTaskSampleHitsPtr)
# define rtmcGetStopRequested(rtmc) (*rtmc->stopRequested)
# define rtmcGetSampleTimePtr(rtmc) (*rtmc->sampleTimes)
# define rtmcGetSampleTimeTaskIDPtr(rtmc) (*rtmc->sampleTimeTaskIDPtr)

# define rtmcGetSampleTime(rtmc,sti) (*rtmc->sampleTimes[sti])

#define rtmcGetTaskTime(rtmc,sti) \
    rtmcGetTPtr(rtmc)[rtmcGetSampleTimeTaskIDPtr(rtmc)[sti]]

/* Only used in SINGLETASKING section of main routine */
#define rtmcIsSampleHit(rtmc,sti,unused) \
    ((rtmcGetSimTimeStep(rtmc) == MAJOR_TIME_STEP) && \
      rtmcGetSampleHitPtr(rtmc)[rtmcGetSampleTimeTaskIDPtr(rtmc)[sti]])

#endif                                  /* _RTW_HEADER_rtmcmacros_h_ */

/* [EOF] rtmcmacros.h */
```
